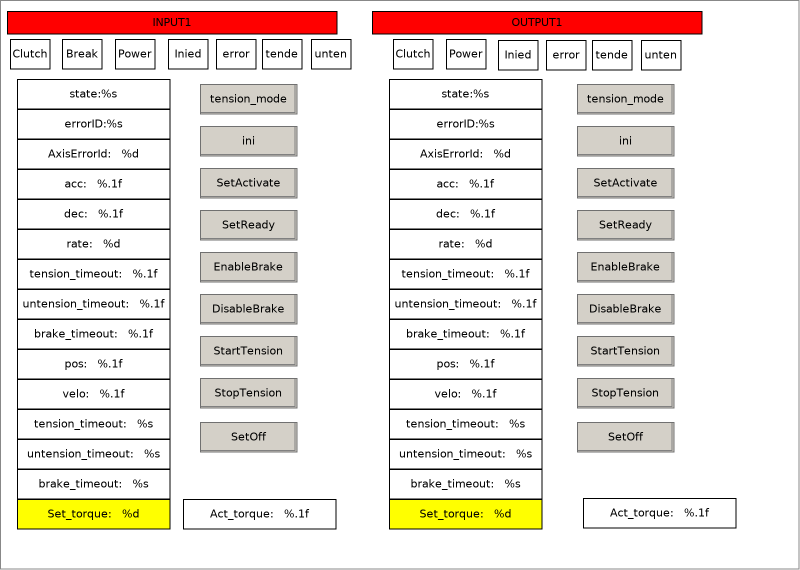
VISUALIZATION VIS_RTR_1  // 800x570
    RoundedRectangle (372,11 330x23), "OUTPUT1"
    RoundedRectangle (7,11 330x23), "INPUT1"
    Button (200,126 97x30), "ini", colour toggle: GVL_API.stRoolToRool[1].Initialize
        toggle GVL_API.stRoolToRool[1].Initialize
    Button (200,84 97x30), "tension_mode", colour toggle: GVL_API.stRoolToRool[1].tension_mode
        toggle GVL_API.stRoolToRool[1].tension_mode
    Button (200,168 97x30), "SetActivate", colour toggle: GVL_API.stRoolToRool[1].SetActivate
        toggle GVL_API.stRoolToRool[1].SetActivate
    Button (200,294 97x30), "DisableBrake", colour toggle: GVL_API.stRoolToRool[1].DisableBrake
        toggle GVL_API.stRoolToRool[1].DisableBrake
    Button (200,210 97x30), "SetReady", colour toggle: GVL_API.stRoolToRool[1].SetReady
        toggle GVL_API.stRoolToRool[1].SetReady
    Button (200,252 97x30), "EnableBrake", colour toggle: GVL_API.stRoolToRool[1].EnableBrake
        toggle GVL_API.stRoolToRool[1].EnableBrake
    Button (200,336 97x30), "StartTension", colour toggle: GVL_API.stRoolToRool[1].StartTension
        toggle GVL_API.stRoolToRool[1].StartTension
    Button (200,378 97x30), "StopTension", colour toggle: GVL_API.stRoolToRool[1].StopTension
        toggle GVL_API.stRoolToRool[1].StopTension
    Button (200,422 97x30), "SetOff", colour toggle: GVL_API.stRoolToRool[1].SetOff
        toggle GVL_API.stRoolToRool[1].SetOff
    RoundedRectangle (62,39 40x30), "Break", colour toggle: stOutput.bqBreakPower[1]
    RoundedRectangle (10,39 40x30), "Clutch", colour toggle: stOutput .bqCluthOut[1]
    Rectangle (17,79 153x30), "state:%s", colour toggle: GVL_API.stRoolToRool[1].state=100, text list: 'TextList_RTRstate', text index: GVL_API.stRoolToRool[1].state
    Rectangle (17,109 153x30), "errorID:%s", colour toggle: GVL_API.stRoolToRool[1].error_code<>0, text list: 'TextList_RTR_errorid', text index: GVL_API.stRoolToRool[1].error_code
    Rectangle (17,169 153x30), "acc: %.1f", text variable: GVL_API.stRoolToRool[1].acceleration
        OnMouseDown: write GVL_API.stRoolToRool[1].acceleration via Default
    Rectangle (17,199 153x30), "dec: %.1f", text variable: GVL_API.stRoolToRool[1].deceleration
        OnMouseDown: write GVL_API.stRoolToRool[1].deceleration via Default
    Rectangle (17,229 153x30), "rate: %d", text variable: GVL_API.stRoolToRool[1].rate
        OnMouseDown: write GVL_API.stRoolToRool[1].rate via Default
    Rectangle (17,259 153x30), "tension_timeout: %.1f", text variable: GVL_API.stRoolToRool[1].tension_timeout
        OnMouseDown: write GVL_API.stRoolToRool[1].tension_timeout via Default
    Rectangle (17,289 153x30), "untension_timeout: %.1f", text variable: GVL_API.stRoolToRool[1].untension_timeout
        OnMouseDown: write GVL_API.stRoolToRool[1].untension_timeout via Default
    Rectangle (17,319 153x30), "brake_timeout: %.1f", text variable: GVL_API.stRoolToRool[1].brake_timeout
        OnMouseDown: write GVL_API.stRoolToRool[1].brake_timeout via Default
    Rectangle (17,139 153x30), "AxisErrorId: %d", text variable: GVL_API.stRoolToRool[1].AxisErrorId
    Rectangle (389,79 153x30), "state:%s", colour toggle: GVL_API.stRoolToRool[2].state=100, text list: 'TextList_RTRstate', text index: GVL_API.stRoolToRool[2].state
    Rectangle (389,109 153x30), "errorID:%s", colour toggle: GVL_API.stRoolToRool[2].error_code<>0, text list: 'TextList_RTR_errorid', text index: GVL_API.stRoolToRool[2].error_code
    Rectangle (389,169 153x30), "acc: %.1f", text variable: GVL_API.stRoolToRool[2].acceleration
        OnMouseDown: write GVL_API.stRoolToRool[2].acceleration via Default
    Rectangle (389,199 153x30), "dec: %.1f", text variable: GVL_API.stRoolToRool[2].deceleration
        OnMouseDown: write GVL_API.stRoolToRool[2].deceleration via Default
    Rectangle (389,229 153x30), "rate: %d", text variable: GVL_API.stRoolToRool[2].rate
        OnMouseDown: write GVL_API.stRoolToRool[2].rate via Default
    Rectangle (389,259 153x30), "tension_timeout: %.1f", text variable: GVL_API.stRoolToRool[2].tension_timeout
        OnMouseDown: write GVL_API.stRoolToRool[2].tension_timeout via Default
    Rectangle (389,289 153x30), "untension_timeout: %.1f", text variable: GVL_API.stRoolToRool[2].untension_timeout
        OnMouseDown: write GVL_API.stRoolToRool[2].untension_timeout via Default
    Rectangle (389,319 153x30), "brake_timeout: %.1f", text variable: GVL_API.stRoolToRool[2].brake_timeout
        OnMouseDown: write GVL_API.stRoolToRool[2].brake_timeout via Default
    Rectangle (389,139 153x30), "AxisErrorId: %d", text variable: GVL_API.stRoolToRool[2].AxisErrorId
    RoundedRectangle (393,39 40x30), "Clutch", colour toggle: stOutput .bqCluthOut[2]
    Button (577,126 97x30), "ini", colour toggle: GVL_API.stRoolToRool[2].Initialize
        toggle GVL_API.stRoolToRool[2].Initialize
    Button (577,84 97x30), "tension_mode", colour toggle: GVL_API.stRoolToRool[2].tension_mode
        toggle GVL_API.stRoolToRool[2].tension_mode
    Button (577,168 97x30), "SetActivate", colour toggle: GVL_API.stRoolToRool[2].SetActivate
        toggle GVL_API.stRoolToRool[2].SetActivate
    Button (577,294 97x30), "DisableBrake", colour toggle: GVL_API.stRoolToRool[2].DisableBrake
        toggle GVL_API.stRoolToRool[1].DisableBrake
    Button (577,210 97x30), "SetReady", colour toggle: GVL_API.stRoolToRool[2].SetReady
        toggle GVL_API.stRoolToRool[2].SetReady
    Button (577,252 97x30), "EnableBrake", colour toggle: GVL_API.stRoolToRool[2].EnableBrake
        toggle GVL_API.stRoolToRool[2].EnableBrake
    Button (577,336 97x30), "StartTension", colour toggle: GVL_API.stRoolToRool[2].StartTension
        toggle GVL_API.stRoolToRool[2].StartTension
    Button (577,378 97x30), "StopTension", colour toggle: GVL_API.stRoolToRool[2].StopTension
        toggle GVL_API.stRoolToRool[2].StopTension
    Button (577,422 97x30), "SetOff", colour toggle: GVL_API.stRoolToRool[2].SetOff
        toggle GVL_API.stRoolToRool[2].SetOff
    RoundedRectangle (115,39 40x30), "Power", colour toggle: P_RollToRoll.FB_RoolToRool[1].REF.Status.ControlLoopClosed
    RoundedRectangle (446,39 40x30), "Power", colour toggle: P_RollToRoll.FB_RoolToRool[2].REF.Status.ControlLoopClosed
    Rectangle (17,349 153x30), "pos: %.1f", text variable: P_RollToRoll.FB_RoolToRool[1].REF.NcToPlc.ActPos
        OnMouseDown: write GVL_API.stRoolToRool[1].brake_timeout via Default
    Rectangle (17,379 153x30), "velo: %.1f", text variable: P_RollToRoll.FB_RoolToRool[1].REF.NcToPlc.ActVelo
        OnMouseDown: write GVL_API.stRoolToRool[1].brake_timeout via Default
    Rectangle (389,349 153x30), "pos: %.1f", text variable: P_RollToRoll.FB_RoolToRool[2].REF.NcToPlc.ActPos
        OnMouseDown: write GVL_API.stRoolToRool[1].brake_timeout via Default
    Rectangle (389,379 153x30), "velo: %.1f", text variable: P_RollToRoll.FB_RoolToRool[2].REF.NcToPlc.ActVelo
        OnMouseDown: write GVL_API.stRoolToRool[1].brake_timeout via Default
    Rectangle (17,409 153x30), "tension_timeout: %s", text variable: P_RollToRoll.FB_RoolToRool[1].tension_ton.ET
    Rectangle (17,439 153x30), "untension_timeout: %s", text variable: P_RollToRoll.FB_RoolToRool[1].untension_ton.ET
    Rectangle (17,469 153x30), "brake_timeout: %s", text variable: P_RollToRoll.FB_RoolToRool[1].enbreak_ton.ET
    Rectangle (389,409 153x30), "tension_timeout: %s", text variable: P_RollToRoll.FB_RoolToRool[2].tension_ton.ET
    Rectangle (389,439 153x30), "untension_timeout: %s", text variable: P_RollToRoll.FB_RoolToRool[2].untension_ton.ET
    Rectangle (389,469 153x30), "brake_timeout: %s", text variable: P_RollToRoll.FB_RoolToRool[2].enbreak_ton.ET
    Rectangle (17,499 153x30), "Set_torque: %d", text variable: HMI_RTR_set_Torque[1]
        OnMouseDown: write HMI_RTR_set_Torque[1] via Default, min 0, max 100
    Rectangle (389,499 153x30), "Set_torque: %d", text variable: HMI_RTR_set_Torque[2]
        OnMouseDown: write HMI_RTR_set_Torque[2] via Default, min 0, max 100
    Rectangle (183,499 153x30), "Act_torque: %.1f", text variable: P_RollToRoll.FB_RoolToRool[1].REF.NcToPlc.ActTorque
    Rectangle (583,498 153x30), "Act_torque: %.1f", text variable: P_RollToRoll.FB_RoolToRool[2].REF.NcToPlc.ActTorque
    RoundedRectangle (168,39 40x30), "Inied", colour toggle: P_RollToRoll.FB_RoolToRool[1].Initialized
    RoundedRectangle (216,39 40x30), "error", colour toggle: P_RollToRoll.FB_RoolToRool[1].error
    RoundedRectangle (262,39 40x30), "tende", colour toggle: P_RollToRoll.FB_RoolToRool[1].tensioned
    RoundedRectangle (311,39 40x30), "unten", colour toggle: P_RollToRoll.FB_RoolToRool[1].untensioned
    RoundedRectangle (498,40 40x30), "Inied", colour toggle: P_RollToRoll.FB_RoolToRool[2].Initialized
    RoundedRectangle (546,40 40x30), "error", colour toggle: P_RollToRoll.FB_RoolToRool[2].error
    RoundedRectangle (592,40 40x30), "tende", colour toggle: P_RollToRoll.FB_RoolToRool[2].tensioned
    RoundedRectangle (641,40 40x30), "unten", colour toggle: P_RollToRoll.FB_RoolToRool[2].untensioned
END_VISUALIZATION

(* stored: Version 1.1.0.1, ProductVersion 3.1.4024.11
   Visu VIS_RTR_1: Id {deb8defa-b467-4469-8e76-dcd47827a96a} *)
